{attribute 'GeneratedUsingTerminal: ELM9410-0000-0016'}
{attribute addProperty BoxType "ELM9410-0000-0016"}
{attribute addProperty Id "ErrorBOOL1UnderrangeBOOL1OverrangeBOOL1DiagBOOL1Sensor_OvrBOOL1OverrunBOOL1TxPDO_StateBOOL1"}
{attribute addProperty CRC "3124567133"}
{attribute addProperty Size "7"}
TYPE Status_BA3D1C5D :
STRUCT
	{attribute addProperty Name "Error"}
	Error : BOOL;
	{attribute addProperty Name "Underrange"}
	Underrange : BOOL;
	{attribute addProperty Name "Overrange"}
	Overrange : BOOL;
	{attribute addProperty Name "Diag"}
	Diag : BOOL;
	{attribute addProperty Name "Sensor_Ovr"}
	Sensor_Ovr : BOOL;
	{attribute addProperty Name "Overrun"}
	Overrun : BOOL;
	{attribute addProperty Name "TxPDO_State"}
	TxPDO_State : BOOL;
END_STRUCT
END_TYPE

(* stored: Version 1.2.0.0, ProductVersion 3.1.4024.9
   DUT Status_BA3D1C5D: Id {2bc60913-4c5b-4b38-a0b9-91c90d0fadd0} *)
